FUNCTION_BLOCK FB_PURGE_N2 EXTENDS FBA_SEQUENCE
VAR_INPUT

END_VAR
VAR_IN_OUT
	Control : TYP_PURGE_N2_CONTROL;
	Parameter: TYP_PURGE_N2_PARAMETER;
END_VAR
VAR_OUTPUT
	Status : TYP_PURGE_N2_STATUS;
END_VAR
VAR
	AlarmHandler : FB_ALARM_HANDLER;
	fbPurgeN2GeneralError : FB_ALARM;
	bInit : BOOL;
	bReset : BOOL;
	bTestalarm : BOOL;
	bTestReset : BOOL;
	bTestAcknowledge : BOOL;
	fbPurgeN2Device : FB_N2_DEVICE;
	State : E_N2_STATES;
END_VAR

//Open valves
//Start purging
//Check if purging time reached
//Repeat x times
//Close valves
//Done := TRUE
IF bInit THEN
	THIS^.Initialize();
	bInit := FALSE;
END_IF

IF bReset THEN
	THIS^.Reset();
	bReset := FALSE;
END_IF

AlarmHandler(Prefix:='PURGE_N2', Repository:=AlarmRepository);
fbPurgeN2GeneralError.Config.Acknowledge := E_ALARM_ACK_TYPE.ACK_AND_RESET;
fbPurgeN2GeneralError.Config.Name := 'PURGE_N2_GENERAL_ERROR';
fbPurgeN2GeneralError.Config.Priority := 3;
fbPurgeN2GeneralError.Config.Code := 1000;
fbPurgeN2GeneralError(Handler := AlarmHandler);

fbPurgeN2Device.AlarmConfig.Name := 'N2_DEVICE';
fbPurgeN2Device.AlarmConfig.Handler REF= AlarmHandler;
fbPurgeN2Device();

//Example how alarms work
IF bTestalarm THEN
	fbPurgeN2GeneralError.Activate();
ELSIF bTestReset THEN
	fbPurgeN2GeneralError.Reset();
ELSIF bTestAcknowledge THEN
	fbPurgeN2GeneralError.Acknowledge();
END_IF

_state(State := State, AlarmHandler := AlarmHandler, StateAsString := TO_STRING(State));

METHOD PUBLIC  Initialize : REFERENCE TO FBA_SEQUENCE
VAR_INPUT
END_VAR
END_METHOD

METHOD PUBLIC  Reset : REFERENCE TO FBA_SEQUENCE
VAR_INPUT
END_VAR
END_METHOD

END_FUNCTION_BLOCK

(* stored: Version 1.1.0.1, ProductVersion 3.1.4024.12
   POU FB_PURGE_N2: Id {c118c864-925d-4c59-b80c-cc2c54f59f1f}, SpecialFunc None
   Method Initialize: Id {25771e6c-3957-489a-a702-edeae513d440}
   Method Reset: Id {ed6229a8-d849-483f-95b8-8ce8abb3a871} *)
